(* PLC project Gen3Safety, BrAutomation SafeDESIGNER  5.19.0.0 *)
(* stored: companyURL http://www.br-automation.com, creationDateTime Wed Apr 10 12:53:51 2024 *)

PROGRAM Main
  VAR  (* added by the conversion: wires and edge detectors of the diagram *)
    _AND_S115_OUT : ANY;
  END_VAR

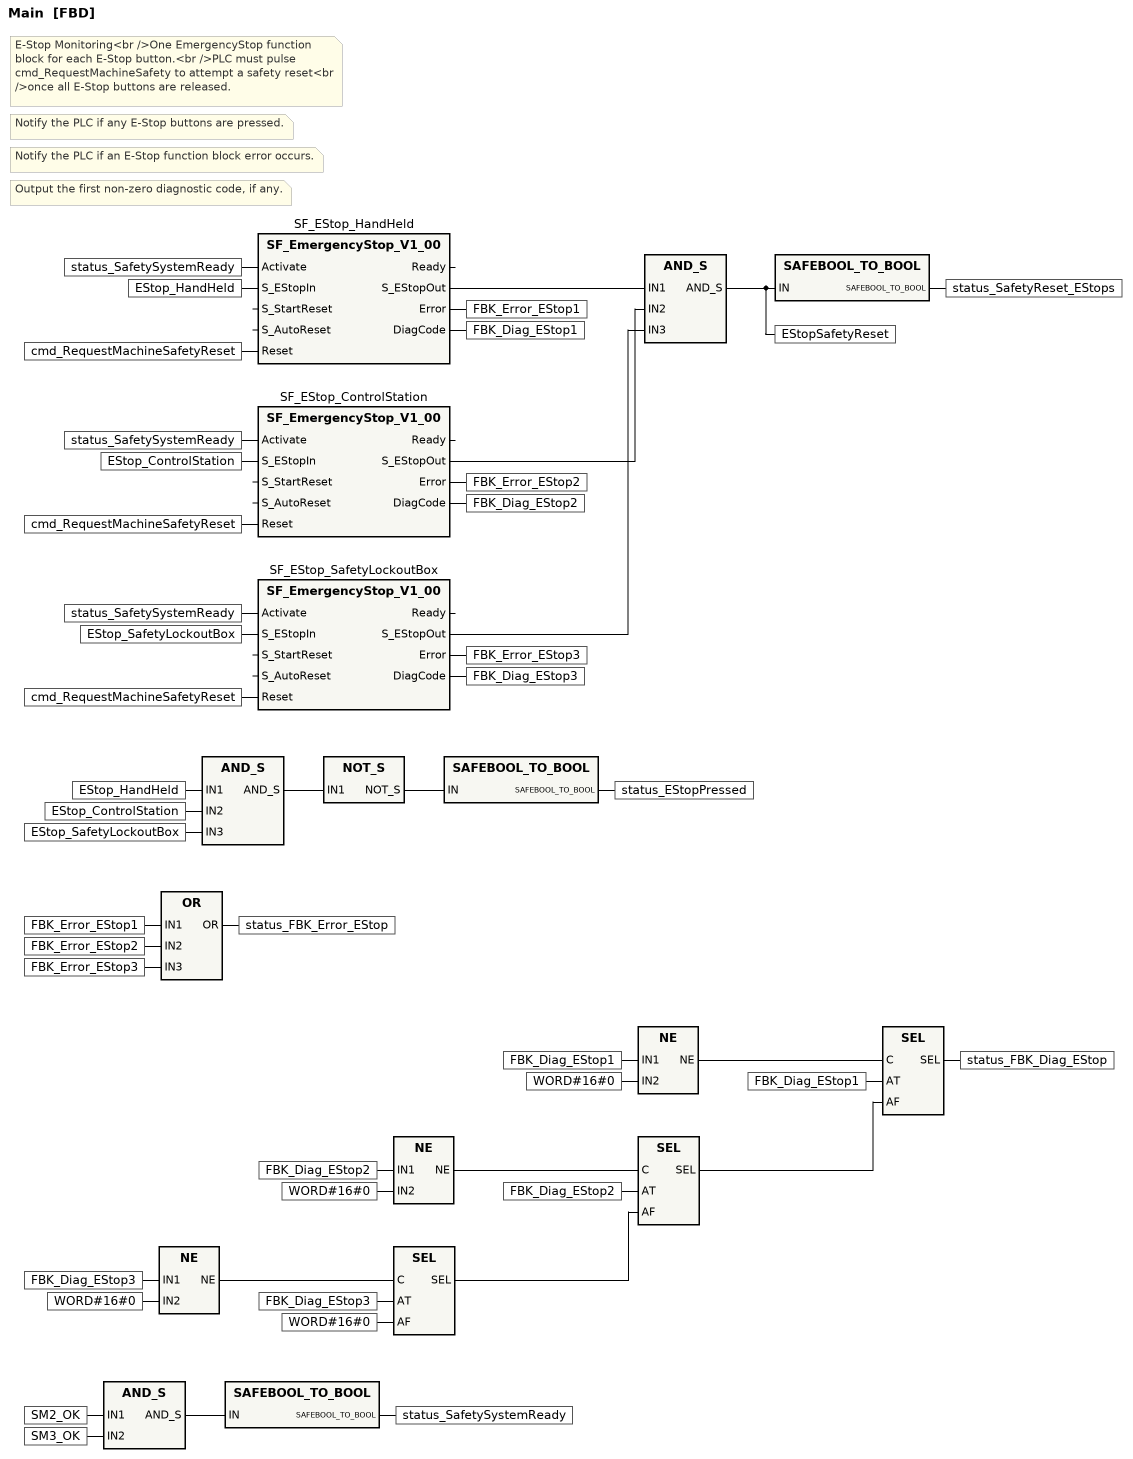
(* FBD diagram, written out as Structured Text *)
(* E-Stop Monitoring<br />One EmergencyStop function block for each E-Stop button.<br />PLC must pulse cmd_RequestMachineSafety to attempt a safety reset<br />once all E-Stop buttons are released. *)
status_SafetySystemReady := SAFEBOOL_TO_BOOL(AND_S(SM2_OK, SM3_OK));
SF_EStop_HandHeld(Activate := status_SafetySystemReady, S_EStopIn := EStop_HandHeld, Reset := cmd_RequestMachineSafetyReset);
FBK_Error_EStop1 := SF_EStop_HandHeld.Error;
FBK_Diag_EStop1 := SF_EStop_HandHeld.DiagCode;
SF_EStop_ControlStation(Activate := status_SafetySystemReady, S_EStopIn := EStop_ControlStation, Reset := cmd_RequestMachineSafetyReset);
SF_EStop_SafetyLockoutBox(Activate := status_SafetySystemReady, S_EStopIn := EStop_SafetyLockoutBox, Reset := cmd_RequestMachineSafetyReset);
_AND_S115_OUT := AND_S(SF_EStop_HandHeld.S_EStopOut, SF_EStop_ControlStation.S_EStopOut, SF_EStop_SafetyLockoutBox.S_EStopOut);
EStopSafetyReset := _AND_S115_OUT;
status_SafetyReset_EStops := SAFEBOOL_TO_BOOL(_AND_S115_OUT);
FBK_Error_EStop2 := SF_EStop_ControlStation.Error;
FBK_Diag_EStop2 := SF_EStop_ControlStation.DiagCode;
FBK_Error_EStop3 := SF_EStop_SafetyLockoutBox.Error;
FBK_Diag_EStop3 := SF_EStop_SafetyLockoutBox.DiagCode;
(* Notify the PLC if any E-Stop buttons are pressed. *)
status_EStopPressed := SAFEBOOL_TO_BOOL(NOT_S(AND_S(EStop_HandHeld, EStop_ControlStation, EStop_SafetyLockoutBox)));
(* Notify the PLC if an E-Stop function block error occurs. *)
status_FBK_Error_EStop := FBK_Error_EStop1 OR FBK_Error_EStop2 OR FBK_Error_EStop3;
(* Output the first non-zero diagnostic code, if any. *)
status_FBK_Diag_EStop := SEL(FBK_Diag_EStop1 <> WORD#16#0, FBK_Diag_EStop1, SEL(FBK_Diag_EStop2 <> WORD#16#0, FBK_Diag_EStop2, SEL(FBK_Diag_EStop3 <> WORD#16#0, FBK_Diag_EStop3, WORD#16#0)));
END_PROGRAM
